// TIA Portal V17 export
// export: Created 2025-03-05T08:02:24.8302687Z, ExportSetting WithDefaults, DisplayName Totally Integrated Automation Portal, DisplayVersion V17 Update 8, DisplayName TIA Portal Openness, DisplayVersion V17 Update 8, DisplayName TIA Portal Version Control Interface, DisplayVersion V17, DisplayName SINAMICS Startdrive Advanced, DisplayVersion V17 SP2, DisplayName SINAMICS Startdrive G110M, G120, G120C, G120D, G120P, G115D, DisplayVersion V17 SP2, DisplayName SINAMICS Startdrive G130, G150, S120, S150, SINAMICS MV, S210, DisplayVersion V17 SP2, DisplayName STEP 7 Professional, DisplayVersion V17 Update 8, DisplayName SINUMERIK ONE STEP 7 Toolbox, DisplayVersion V17 Update 12, DisplayName SINUMERIK 840D sl STEP 7 Toolbox, DisplayVersion V17 Update 12, DisplayName STEP 7 Safety, DisplayVersion V17 Update 6, DisplayName WinCC Advanced, DisplayVersion V17 Update 8
TYPE "INTERLOCKS_ETXETAR_ROBOT_CELL_GENERAL"
// stored: IsFailsafeCompliant false
   STRUCT
      MACHINE_TO_CELL : Struct
         MCH_MEAS_STA_CALIBRATION_REQ : Bool;   // MACHINE MEAS STATION CALIBRATION REQUIRED
         MCH_MEAS_STA_READY_TO_MEASURE : Bool;   // MACHINE MEAS STATION READY TO MEASURE
         MCH_MEAS_STA_MEASURE_IN_PRCESS : Bool;   // MACHINE MEAS STATION MEASUREMENT IN PROCESS
         MCH_MEAS_STA_MEASURE_FINISHED : Bool;   // MACHINE MEAS STATION MEASUREMENT FINISHED
         MCH_MEAS_STA_HOME_POSITION : Bool;   // MACHINE MEAS STATION AT HOME POSITION
         MCH_MEAS_STA_FAULT : Bool;   // MACHINE MEAS STATION FAULT
         PNEUMATIC_IN_SERVICE_SPARE_0_5 : Bool;
         SPARE_0_7 : Bool;
         MCH_MEAS_STA_MICROEPSILON_FACE_R_ENABLED : Bool;   // MACHINE MEAS STATION MICROEPSILON FACE R ENABLED
         MCH_MEAS_STA_MICROEPSILON_FACE_N_ENABLED : Bool;   // MACHINE MEAS STATION MICROEPSILON FACE N ENABLED
         SPARE_1_2 : Bool;
         SPARE_1_3 : Bool;
         SPARE_1_4 : Bool;
         SPARE_1_5 : Bool;
         SPARE_1_6 : Bool;
         SPARE_1_7 : Bool;
         SPARE_MEAS_STA : Array[0..5] of Byte;
         COOLING_SPARE : Bool;
         SPARE_8_1 : Bool;
         SPARE_8_2 : Bool;
         SPARE_8_3 : Bool;
         SPARE_8_4 : Bool;
         SPARE_8_5 : Bool;
         SPARE_8_6 : Bool;
         SPARE_8_7 : Bool;
         SPARE_9_0 : Bool;
         SPARE_9_1 : Bool;
         SPARE_9_2 : Bool;
         SPARE_9_3 : Bool;
         SPARE_9_4 : Bool;
         SPARE_9_5 : Bool;
         SPARE_9_6 : Bool;
         SPARE_9_7 : Bool;
         SPARE_COOLING : Array[0..5] of Byte;
         MCH_EKS_CURRENT_PROTECTION_LVL : Byte;   // MACHINE EKS CURRENT ACCESS LEVEL
         MCH_EKS_IDENT_1 : Byte;   // MACHINE EKS OPERATOR ID CHAR 1
         MCH_EKS_IDENT_2 : Byte;   // MACHINE EKS OPERATOR ID CHAR 2
         MCH_EKS_IDENT_3 : Byte;   // MACHINE EKS OPERATOR ID CHAR 3
         MCH_EKS_IDENT_4 : Byte;   // MACHINE EKS OPERATOR ID CHAR 4
         MCH_EKS_IDENT_5 : Byte;   // MACHINE EKS OPERATOR ID CHAR 5
         MCH_EKS_IDENT_6 : Byte;   // MACHINE EKS OPERATOR ID CHAR 6
         MCH_EKS_IDENT_7 : Byte;   // MACHINE EKS OPERATOR ID CHAR 7
         MCH_EKS_IDENT_8 : Byte;   // MACHINE EKS OPERATOR ID CHAR 8
         MCH_EKS_OPERATOR_IDENTIFICATION : Byte;   // MACHINE EKS OPERATOR IDENTIFICATION
         SPARE_26_0 : Bool;
         SPARE_26_1 : Bool;
         SPARE_26_2 : Bool;
         SPARE_26_3 : Bool;
         SPARE_26_4 : Bool;
         SPARE_26_5 : Bool;
         SPARE_26_6 : Bool;
         SPARE_26_7 : Bool;
         SPARE_27_0 : Bool;
         SPARE_27_1 : Bool;
         SPARE_27_2 : Bool;
         SPARE_27_3 : Bool;
         SPARE_27_4 : Bool;
         SPARE_27_5 : Bool;
         SPARE_27_6 : Bool;
         SPARE_27_7 : Bool;
         SPARE_GENERAL : Array[0..34] of Byte;
      END_STRUCT;
      CELL_TO_MACHINE : Struct
         CELL_MEAS_STA_START_MEAS_CYCLE : Bool;   // CELL MEASURING STATION START MEASURING CYCLE
         CELL_MEAS_STA_START_CALIB_CYCLE : Bool;   // CELL MEASURING STATION START CALIBRATION CYCLE
         CELL_MEAS_STA_HOME_REQ : Bool;   // CELL MEASURING STATION HOME REQUEST
         CELL_MEAS_STA_FAULT : Bool;   // CELL MEASURING STATION FAULT
         CELL_MEAS_STA_RESET : Bool;   // CELL MEASURING STATION RESET
         CALIB_MODE_SLCTD_SPARE_0_5 : Bool;
         SPARE_0_6 : Bool;
         SPARE_0_7 : Bool;
         CELL_MEAS_STA_PART_LOADED : Bool;   // CELL MEASURING STATION PART LOADED
         CELL_MEAS_STA_PART_UNLOADED : Bool;   // CELL MEASURING STATION PART UNLOADED
         SPARE_1_2 : Bool;
         SPARE_1_3 : Bool;
         SPARE_1_4 : Bool;
         SPARE_1_5 : Bool;
         SPARE_1_6 : Bool;
         SPARE_1_7 : Bool;
         SPARE_MEAS_STA : Array[0..5] of Byte;
         CELL_COOLING_DEGRADED_MODE : Bool;   // CELL COOLING DEGRADED MODE
         SPARE_8_1 : Bool;
         SPARE_8_2 : Bool;
         SPARE_8_3 : Bool;
         SPARE_8_4 : Bool;
         SPARE_8_5 : Bool;
         SPARE_8_6 : Bool;
         SPARE_8_7 : Bool;
         SPARE_9_0 : Bool;
         SPARE_9_1 : Bool;
         SPARE_9_2 : Bool;
         SPARE_9_3 : Bool;
         SPARE_9_4 : Bool;
         SPARE_9_5 : Bool;
         SPARE_9_6 : Bool;
         SPARE_9_7 : Bool;
         SPARE_COOLING : Array[0..5] of Byte;
         CELL_STARVED : Bool;   // CELL STARVED
         CELL_BLOCKED : Bool;   // CELL BLOCKED
         SPARE_16_2 : Bool;
         SPARE_16_3 : Bool;
         SPARE_16_4 : Bool;
         SPARE_16_5 : Bool;
         SPARE_16_6 : Bool;
         SPARE_16_7 : Bool;
         SPARE_17_0 : Bool;
         SPARE_17_1 : Bool;
         SPARE_17_2 : Bool;
         SPARE_17_3 : Bool;
         SPARE_17_4 : Bool;
         SPARE_17_5 : Bool;
         SPARE_17_6 : Bool;
         SPARE_17_7 : Bool;
         SPARE_GENERAL : Array[0..45] of Byte;
      END_STRUCT;
   END_STRUCT;
END_TYPE
